// TIA Portal V19 export
TYPE "PPrf_SetUp_Man"
// stored: Access Published
   STRUCT
      X : Array[1.."SET_UP_MAN_ADJUST_MAX"] of Real;
      Y : Array[1.."SETUP_MAN_OP_WITH_CODE_QTY"] of Int;
   END_STRUCT;
END_TYPE
